{attribute 'enable_dynamic_creation'}	
{attribute 'no_explicit_call' := 'do not call this function block directly'} 
FUNCTION_BLOCK FileReadStringTask EXTENDS FileContentTask
VAR
	_ClassName : STRING := __POUNAME();

	_ReadString : Tc2_System.FB_FileGets;
END_VAR

{attribute 'monitoring' := 'call'}
PROPERTY ClassName : STRING
GET
ClassName := _ClassName;
END_GET
END_PROPERTY

METHOD Execute : BOOL
VAR_INPUT
	start : BOOL;
END_VAR
IF start THEN
	Validate();

	_ReadString(
		bExecute := FALSE,
		hFile := FilecontentManager.FileHandle,
		sNetId := FilecontentManager.AmsNetId,
		tTimeout := Timeout
	);	
END_IF

_ReadString(bExecute := TRUE);

IF _ReadString.bError THEN
	//exceptionFactory.ThrowException(__POSITION(), WStringHelper.Concat2("Read string from file failed", GetErrorMessageByErrorId(_ReadString.nErrId)), __POUNAME(), ClassName, CurrentNamespace.Name, __POSITION(), _ReadString.nErrId);
ELSIF NOT _ReadString.bBusy THEN
	Execute := EXECUTION_STATE.DONE;
END_IF
END_METHOD

PROPERTY LoadedString : REFERENCE TO Tc2_System.T_MaxString
GET
LoadedString REF= _ReadString.sLine;
END_GET
END_PROPERTY

METHOD PROTECTED Validate
SUPER^.Validate();

CASE FileContentManager.OpenMode OF
	FILE_OPEN_MODE.APPEND, FILE_OPEN_MODE.WRITE_EMPTY:
		//exceptionFactory.ThrowException(__POSITION(), "File is not open for reading");
END_CASE

IF FileContentManager.ContentHandlingMode <> FILE_CONTENT_HANDLING_MODE.TEXT THEN
	//exceptionFactory.ThrowException(__POSITION(), "File is not open in text mode");
END_IF
END_METHOD

END_FUNCTION_BLOCK

(* stored: Version 1.1.0.1
   POU FileReadStringTask: Id {50658161-f2b3-4754-8024-f8b761c7e377}, SpecialFunc None
   Property ClassName: Id {17e8b6c3-5b1c-47e7-86d9-eb28eb0dd80c}
   Get Get: Id {d086ac05-b4a6-44fc-9822-2f644494f311}
   Method Execute: Id {669cb495-c528-4127-9fbd-46ab13f9f858}
   Property LoadedString: Id {8e690dbc-86bf-4f83-9be8-37ea8a152b00}
   Get Get: Id {cffff10f-c614-4c56-932d-c14bb2781531}
   Method Validate: Id {8929b0fb-3ef1-4c4c-b56e-e2bd279a7458} *)
